PROGRAM MAIN_simu
VAR
	simIO: MNG_Simulation;
	outputs: MNG_Application_Outputs_32Bit;
	inputs: MNG_Application_Inputs_32Bit;
	//ioUpdater: MNG_UpdateIOs := (sRemoteHost := '192.168.192.115', nRemotePort := 5000);
	
	bEnable: BOOL := TRUE;
	
	i: INT;
	fbIOLink	: FB_IOLink;
END_VAR

VAR_INPUT
	bExecute: BOOL;
END_VAR

// Update IOs with simulation

simIO(bEnable := bEnable, outputs := outputs, inputs => inputs);

// Mapping of the IO´s

fbIOLink(goon := TRUE, inputs := inputs, outputs => outputs);

END_PROGRAM

(* stored: Version 1.1.0.1, ProductVersion 3.1.0.25
   POU MAIN_simu: Id {5a30d4c3-f2cc-4a3c-9111-ebd3bd8d2e80} *)
